// LS Electric XG5000 project: 사칙연산
// PLC LSPLC
// module base 0 slot 0: 입출력 모듈:XBC-DR14E (DC 24V 입력 8점, 릴레이 출력 6점)

PROGRAM NewProgram (task: 스캔 프로그램)

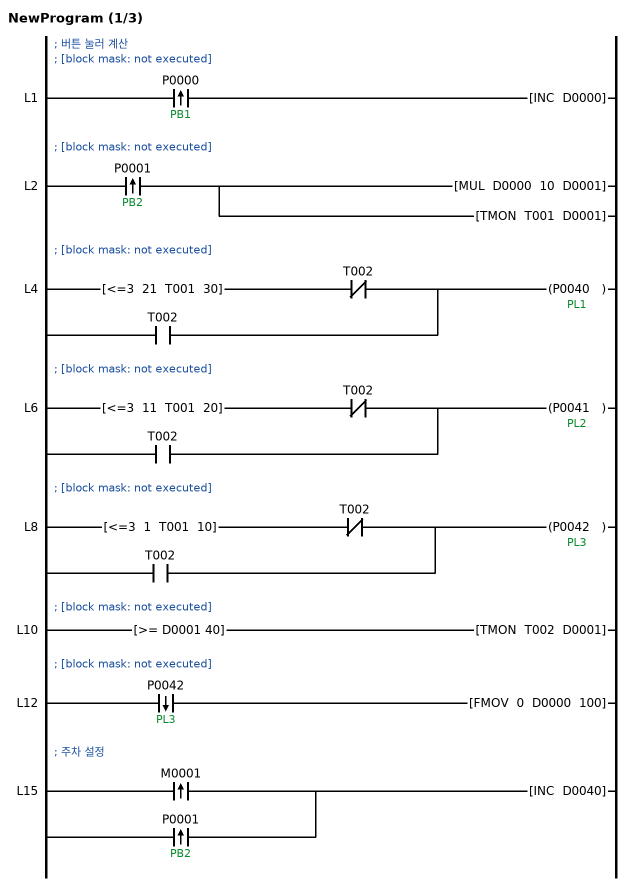
// 버튼 눌러 계산
; L1 (block mask: not executed)
LOADP     P0000	// PB1
INC       D0000
; L2 (block mask: not executed)
LOADP     P0001	// PB2
MUL       D0000 10 D0001
TMON      T001 D0001
; L4 (block mask: not executed)
LOAD<=3   21 T001 30
AND NOT   T002
OR        T002
OUT       P0040	// PL1
; L6 (block mask: not executed)
LOAD<=3   11 T001 20
AND NOT   T002
OR        T002
OUT       P0041	// PL2
; L8 (block mask: not executed)
LOAD<=3   1 T001 10
AND NOT   T002
OR        T002
OUT       P0042	// PL3
; L10 (block mask: not executed)
LOAD>=    D0001 40
TMON      T002 D0001
; L12 (block mask: not executed)
LOADN     P0042	// PL3
FMOV      0 D0000 100
// 주차 설정
; L15
LOADP     M0001
ORP       P0001	// PB2
INC       D0040

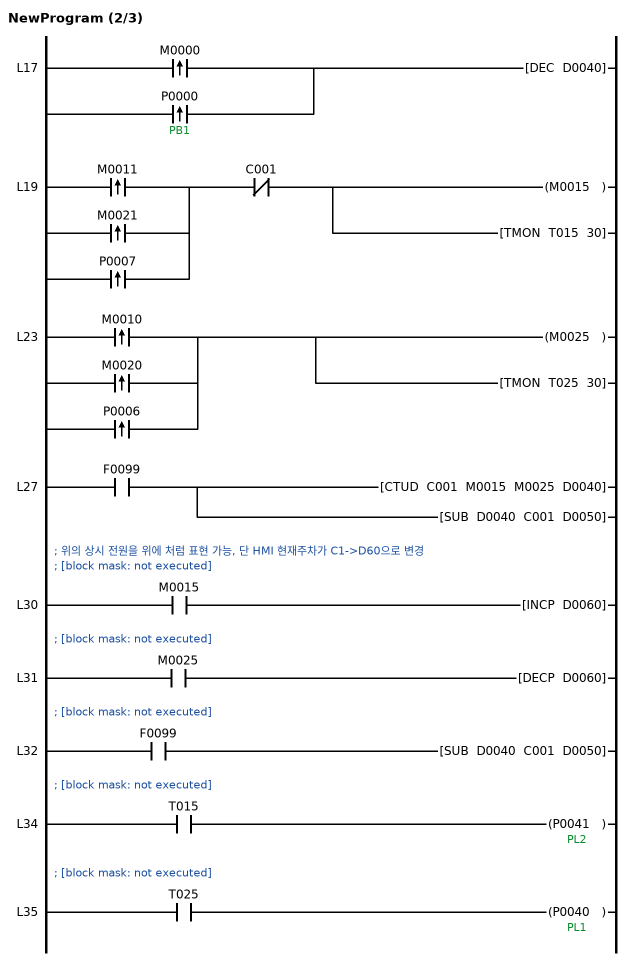
; L17
LOADP     M0000
ORP       P0000	// PB1
DEC       D0040
; L19
LOADP     M0011
ORP       M0021
ORP       P0007
AND NOT   C001
OUT       M0015
TMON      T015 30
; L23
LOADP     M0010
ORP       M0020
ORP       P0006
OUT       M0025
TMON      T025 30
; L27
LOAD      F0099
CTUD      C001 M0015 M0025 D0040
SUB       D0040 C001 D0050
// 위의 상시 전원을 위에 처럼 표현 가능, 단 HMI 현재주차가 C1->D60으로 변경
; L30 (block mask: not executed)
LOAD      M0015
INCP      D0060
; L31 (block mask: not executed)
LOAD      M0025
DECP      D0060
; L32 (block mask: not executed)
LOAD      F0099
SUB       D0040 C001 D0050
; L34 (block mask: not executed)
LOAD      T015
OUT       P0041	// PL2
; L35 (block mask: not executed)
LOAD      T025
OUT       P0040	// PL1

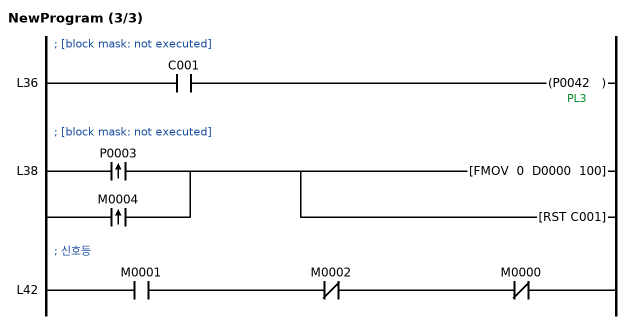
; L36 (block mask: not executed)
LOAD      C001
OUT       P0042	// PL3
; L38 (block mask: not executed)
LOADP     P0003
ORP       M0004
FMOV      0 D0000 100
RST       C001
// 신호등
; L42
LOAD      M0001
AND NOT   M0002
AND NOT   M0000

VARIABLES AND COMMENTS (devices not used above)
P00002	BIT	PB3
P00043	BIT	PL4